FUNCTION_BLOCK FB_DoWork

METHOD M_ConsumeTime : Global.HRESULT
VAR_INPUT
	CallerTaskAdsPort : UINT;
END_VAR

VAR_INST
	fbRTMon_LogMark : FB_RTMon_LogMark;
END_VAR
fbRTMon_LogMark.LogStart(CallerTaskAdsPort, 0);
F_ConsumeTime(100);
fbRTMon_LogMark.LogStop(CallerTaskAdsPort, 0);
END_METHOD

END_FUNCTION_BLOCK

(* stored: Version 1.1.0.1, ProductVersion 3.1.4026.18
   POU FB_DoWork: Id {fdd8d320-d86d-45ca-89fd-e20a01bfe114}, SpecialFunc None
   Method M_ConsumeTime: Id {57505c6f-4d23-40e1-aa82-1354117ea6a0} *)
